(* CoDeSys 2.3.9.13 project: Stepper_03_Example02.pro *)
(* Libraries: D:\Daten\CodeSys_841\Projekte\Stepper\MC3\Release0.9.2\Stepper_03.lib 9.7.09 14:06:03, Standard.lib 22.11.04 11:21:12 *)

(* PLC configuration (modules and I/O channels)
Module Fieldbus Assignment [WAGO_Module] node 0, in %IB0 out %QB0 {INTTypePAAssignment = PLC; INTTypeModule = plugged}
Module Fieldbus Assignment [WAGO_Module] node 1, in %IB1 out %QB1 {INTTypePAAssignment = PLC; INTTypeModule = plugged}
Fieldbus variables [FB_VARS] node 1, in %IB0 out %QB0
*)

(* POU PLC_PRG, FBD *)
PROGRAM PLC_PRG
VAR

	myconfigtest673				:MC3_typConfiguration_673;

	Stepper1In AT%IB0			: ARRAY[0..11] OF BYTE;		(* input address stepper modul 750-673 *)
	Stepper1Out  AT%QB0 		: ARRAY[0..11] OF BYTE;		(* output address stepper modul 750-673 *)

	data1							: MC3_typData;
	MyCT							: MC3_ConfigurationTable;
	executeCT						: BOOL;
	readCT						: BOOL;
	writeCT						: BOOL;
	doneCT						: BOOL;
	busyCT						: BOOL;
	errorCT						: BOOL;
	statusCT						: WORD;

	MyDPT							: MC3_DriveProgramTable;
	executeDPT					: BOOL;
	readDPT						: BOOL;
	writeDPT						: BOOL;
	flashprogramDPT				: BOOL;
	dataCountDPT				: WORD:=14;
	doneDPT						: BOOL;
	busyDPT						: BOOL;
	errorDPT						: BOOL;
	statusDPT						: WORD;
	DataDPT		: ARRAY [0..MC3_gc_DriveProgramTableSize] OF BYTE:=
	(* opcode,  data_LSB, data, data_MSB  *)
		16#25, 16#20, 16#4E, 16#00,			(* set velocity  to 20.000 *)
		16#22, 16#B8, 16#0B, 16#00,			(* set acceleration to 3.000 *)
		16#04, 16#02, 16#00, 16#00,			(* Move_L to position 2 from position table*)
		16#70, 16#D0, 16#07, 16#00,			(* wait 2000 ms *)
		16#06, 16#88, 16#C3, 16#00,			(* Move relative 5.000 *)
		16#70, 16#D0, 16#07, 16#00,			(* wait 2000 ms *)
		16#06, 16#88, 16#C3, 16#00,			(* Move relative 5.000 *)
		16#70, 16#D0, 16#07, 16#00,			(* wait 2000 ms *)
		16#06, 16#88, 16#C3, 16#00,			(* Move relative 5.000 *)
		16#70, 16#D0, 16#07, 16#00,			(* wait 2000 ms *)
		16#25, 16#10, 16#27, 16#00,			(* set velocity to 10.000 *)
		16#02, 16#00, 16#00, 16#00,			(* move to position 0 *)
		16#02, 16#00, 16#00, 16#00,			(* move to position 0 *)
		16#F1, 16#00, 16#00, 16#00;			(* end, wenn das Fahrprogramm hiermit abgeschlossen wird, gibt es keinen Fehler am Ende *)

	PositionTable					: ARRAY [0..MC3_gc_PositionTableSize] OF BYTE:=
	(*  data_LSB, data, data_MSB  *)
		16#00, 16#10, 16#00, 16#00,			(* Position 0->8192 *)
		16#00, 16#20, 16#00, 16#00,			(* Position 1->16384 *)
		16#A0, 16#86, 16#01, 16#00,			(* Position 2->100.000*)
		16#C0, 16#D4, 16#01, 16#00;			(* Position 3->120.000*)
	executePT					: BOOL;
	readPT						: BOOL;
	writePT						: BOOL;
	dataCountPT				: BYTE:=4;


	donePT						: BOOL;
	busyPT						: BOOL;
	errorPT						: BOOL;
	statusPT						: WORD;

	MyJog672						: MC3_Jog_672;
	enableJOG					: BOOL;
	TimeoutJOG					: WORD;
	busyJOG						: BOOL;

	MyMoveRelative				: MC3_MoveRelative;
	executeMoveRelative			: BOOL;
	SpeedMoveRelative			: INT:=10000;
	AccelerationMoveRelative		: WORD:=32000;
	DecelerationMoveRelative	: WORD:=32000;
	PositionMoveRelative			: DINT:=100000;
	doneMoveRelative			: BOOL;
	busyMoveRelative				: BOOL;
	errorMoveRelative				: BOOL;


	MyMoveAbsolute				: MC3_MoveAbsolute;
	executeMoveAbsolute			: BOOL;
	SpeedMoveAbsolute			: INT:=10000;
	AccelerationMoveAbsolute	: WORD:=30000;
	PositionMoveAbsolute		: DINT:=20000;
	busyMoveAbsolute			: BOOL;
	doneMoveAbsolute			: BOOL;

	MyHoming						: MC3_Home;
	executeHoming				: BOOL;
	HomingPositive				: BOOL;
	HomingNegative				: BOOL;
	doneHoming					: BOOL;
	busyHoming					: BOOL;

	MyVelocity672					: MC3_MoveVelocity_672;
	executeMoveVelocity			: BOOL;
	SpeedMoveVelocity			: INT;
	AccelerationMoveVelocity		: WORD:=200;
	doneMoveVelocity				: BOOL;
	busyMoveVelocity				: BOOL;

	MyPower						: MC3_Power;
	enablePower					: BOOL;
	PowerEnabled				: BOOL;

	MyReadActualPosition		: MC3_ReadActualPosition;
	enableRead					: BOOL:=TRUE;
	PositionValid					: BOOL;
	ActualPosition					: DINT;
	ActualSpeed					: INT;
	ActualMode					: BYTE;
	MailboxActive					: BOOL;
	ModulReset					: BOOL;

	MyReset						: MC3_Reset;
	executeReset					: BOOL;
	doneReset					: BOOL;

	MyStop							: MC3_Stop;
	executeStop					: BOOL;
	doneStop						: BOOL;

	MyReadError					: MC3_ReadError;
	enableReadError				: BOOL;
	doneReadError				: BOOL;
	busyReadError				: BOOL;
	StepperError					: BOOL;
	status							: WORD;
	ErrorDescription				: MC3_error_codes;

	MySetPosition					: MC3_SetPosition;
	executeSet					: BOOL;
	positionSet					: DINT;
	doneSet						: BOOL;
	busySet						: BOOL;
	errorSet						: BOOL;

	MyDP							: MC3_DriveProgram;
	executeDP						: BOOL;
	startpositionDP				: WORD;
	doneDP						: BOOL;
	busyDP						: BOOL;
	actualpositionDP				: WORD;

	MyCV							: MC3_ConfigurationValue;
	executeCV						: BOOL;
	addressCV					: WORD;
	readwriteCV					: BYTE;
	valuesizeCV					: BYTE;
	valueCV						: DWORD;
	doneCV						: BOOL;
	busyCV						: BOOL;
	errorCV						: BOOL;
	statusCV						: WORD;



(*visualisation variables*)
	visu_enablePower:BOOL;
	visu_executeReset:BOOL;
	(*Basic_1: MC2_StepperControlBasic;
	BasicEnable: BOOL;
	BasicDone: BOOL;
	BasicJobType: MC2_Mode;
	BasicModule: WORD:=670;
	BasicPos: BOOL;
	BasicNeg: BOOL;
	BasicStop: BOOL;
	BasicSpeed: INT:=5000;
	BasicAcceleration: WORD:=10000;
	BasicDeceleration: WORD:=10000;
	BasicRefPosition: DINT:=100000;
	BasicStart: BOOL;
	BasicReset: BOOL;
	BasicBusy: BOOL;
	BasicActualPosition: DINT;
	BasicActualSpeed: INT;
	BasicMailboxActive: BOOL;
	BasicError: BOOL;
	BasicStatus: WORD;
	BasicErrorCodes: MC2_Error_Codes;*)
	startablauf: BOOL;
	ablaufstate: INT;

	count: INT;
	testcount: INT := 1;
	MyVelocity670: MC3_MoveVelocity_670;
	MyJog670: MC3_Jog_670;
	posJog: BOOL;
	negJog: BOOL;

	executeDefault: BOOL;
	doneDefault: BOOL;
	busyDefault: BOOL;
	errorDefault: BOOL;
	StatusDefault: WORD;
	Stepper_673: MC3_StepperCommunication;
	P3: MC3_Power;
	S3: MC3_Stop;
	R3: MC3_MoveRelative;
	M3: MC3_Home;
	Re3: MC3_Reset;
	Abs3: MC3_MoveAbsolute;
	MySetPosition3: MC3_SetPosition;
	MyReadActualPosition3: MC3_ReadActualPosition;
	MyReadError3: MC3_ReadError;
	MyCT3: MC3_ConfigurationTable;
	MyCV3: MC3_ConfigurationValue;
	MyVelocity672_3: MC3_MoveVelocity_672;
	MyJog670_3: MC3_Jog_672;
	jogTimeout: WORD;
	b1: MC3_StepperControlBasic;
	error: BOOL;
	TON1: TON;
	testwert1: DINT;
	Torque3: MC3_MoveTorque;
	doneTorque: BOOL;
	busyTorque: BOOL;
	executeTorque: BOOL;
	speedTorque: INT;
	currentTorque: WORD;
	Torque3_2: MC3_MoveTorque2;
	enableTorque: BOOL;
	doneTorque2: BOOL;
	busyTorque2: BOOL;
	MyDT: MC3_DriveProgramTable;
	MyPT: MC3_PositionTable;
	MyVelocity670_3: MC3_MoveVelocity_670;
	MyJog672_3: MC3_Jog_672;
END_VAR
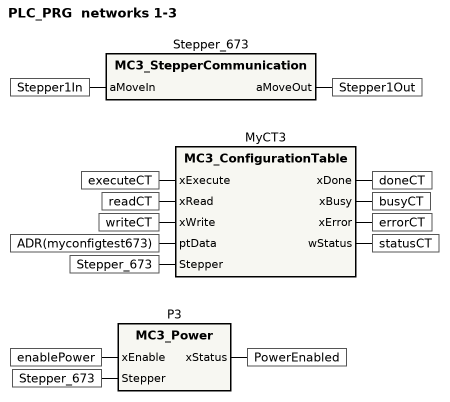
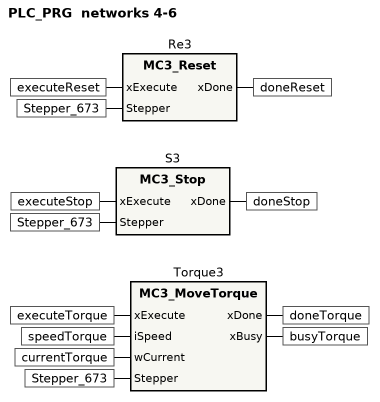
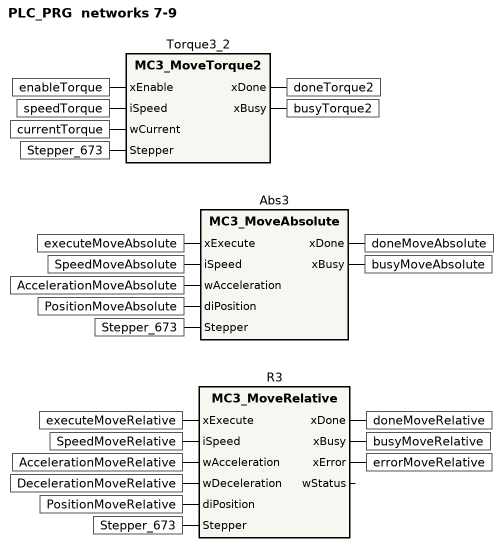
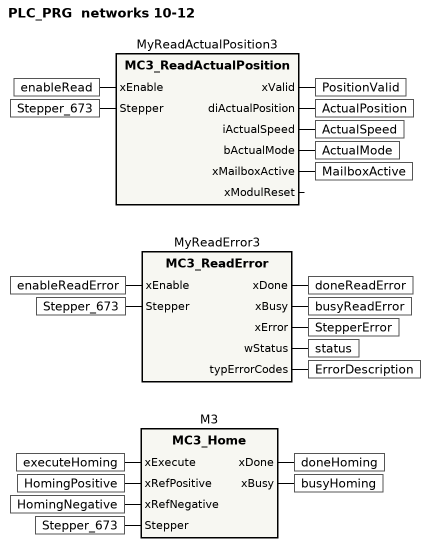
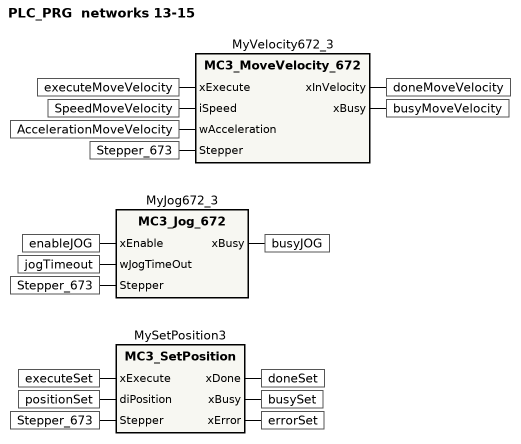
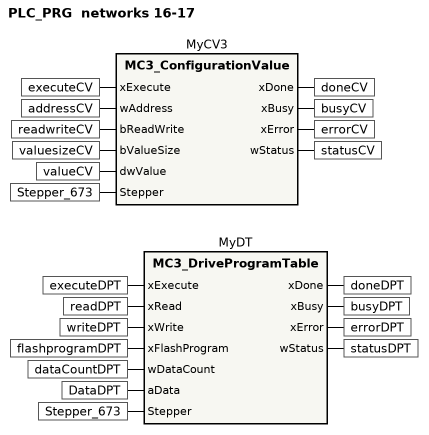
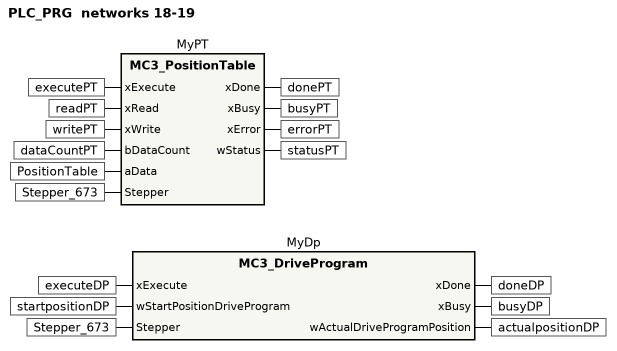
_FBD_ (* Function Block Diagram *)
NETWORK 1
	Stepper_673:MC3_StepperCommunication(aMoveIn: Stepper1In) => Stepper1Out
NETWORK 2
	MyCT3:MC3_ConfigurationTable(xExecute: executeCT, xRead: readCT, xWrite: writeCT, ptData: ADR(myconfigtest673), Stepper: Stepper_673, xBusy => busyCT, xError => errorCT, wStatus => statusCT) => doneCT
NETWORK 3
	P3:MC3_Power(xEnable: enablePower, Stepper: Stepper_673) => PowerEnabled
NETWORK 4
	Re3:MC3_Reset(xExecute: executeReset, Stepper: Stepper_673) => doneReset
NETWORK 5
	S3:MC3_Stop(xExecute: executeStop, Stepper: Stepper_673) => doneStop
NETWORK 6
	Torque3:MC3_MoveTorque(xExecute: executeTorque, iSpeed: speedTorque, wCurrent: currentTorque, Stepper: Stepper_673, xBusy => busyTorque) => doneTorque
NETWORK 7
	Torque3_2:MC3_MoveTorque2(xEnable: enableTorque, iSpeed: speedTorque, wCurrent: currentTorque, Stepper: Stepper_673, xBusy => busyTorque2) => doneTorque2
NETWORK 8
	Abs3:MC3_MoveAbsolute(xExecute: executeMoveAbsolute, iSpeed: SpeedMoveAbsolute, wAcceleration: AccelerationMoveAbsolute, diPosition: PositionMoveAbsolute, Stepper: Stepper_673, xBusy => busyMoveAbsolute) => doneMoveAbsolute
NETWORK 9
	R3:MC3_MoveRelative(xExecute: executeMoveRelative, iSpeed: SpeedMoveRelative, wAcceleration: AccelerationMoveRelative, wDeceleration: DecelerationMoveRelative, diPosition: PositionMoveRelative, Stepper: Stepper_673, xBusy => busyMoveRelative, xError => errorMoveRelative) => doneMoveRelative
NETWORK 10
	MyReadActualPosition3:MC3_ReadActualPosition(xEnable: enableRead, Stepper: Stepper_673, diActualPosition => ActualPosition, iActualSpeed => ActualSpeed, bActualMode => ActualMode, xMailboxActive => MailboxActive) => PositionValid
NETWORK 11
	MyReadError3:MC3_ReadError(xEnable: enableReadError, Stepper: Stepper_673, xBusy => busyReadError, xError => StepperError, wStatus => status, typErrorCodes => ErrorDescription) => doneReadError
NETWORK 12
	M3:MC3_Home(xExecute: executeHoming, xRefPositive: HomingPositive, xRefNegative: HomingNegative, Stepper: Stepper_673, xBusy => busyHoming) => doneHoming
NETWORK 13
	MyVelocity672_3:MC3_MoveVelocity_672(xExecute: executeMoveVelocity, iSpeed: SpeedMoveVelocity, wAcceleration: AccelerationMoveVelocity, Stepper: Stepper_673, xBusy => busyMoveVelocity) => doneMoveVelocity
NETWORK 14
	MyJog672_3:MC3_Jog_672(xEnable: enableJOG, wJogTimeOut: jogTimeout, Stepper: Stepper_673) => busyJOG
NETWORK 15
	MySetPosition3:MC3_SetPosition(xExecute: executeSet, diPosition: positionSet, Stepper: Stepper_673, xBusy => busySet, xError => errorSet) => doneSet
NETWORK 16
	MyCV3:MC3_ConfigurationValue(xExecute: executeCV, wAddress: addressCV, bReadWrite: readwriteCV, bValueSize: valuesizeCV, dwValue: valueCV, Stepper: Stepper_673, xBusy => busyCV, xError => errorCV, wStatus => statusCV) => doneCV
NETWORK 17
	MyDT:MC3_DriveProgramTable(xExecute: executeDPT, xRead: readDPT, xWrite: writeDPT, xFlashProgram: flashprogramDPT, wDataCount: dataCountDPT, aData: DataDPT, Stepper: Stepper_673, xBusy => busyDPT, xError => errorDPT, wStatus => statusDPT) => doneDPT
NETWORK 18
	MyPT:MC3_PositionTable(xExecute: executePT, xRead: readPT, xWrite: writePT, bDataCount: dataCountPT, aData: PositionTable, Stepper: Stepper_673, xBusy => busyPT, xError => errorPT, wStatus => statusPT) => donePT
NETWORK 19
	MyDp:MC3_DriveProgram(xExecute: executeDP, wStartPositionDriveProgram: startpositionDP, Stepper: Stepper_673, xBusy => busyDP, wActualDriveProgramPosition => actualpositionDP) => doneDP
_END_FBD_
(* the same logic as Structured Text *)
(* Network 1 *)
Stepper_673(aMoveIn := Stepper1In);
Stepper1Out := Stepper_673.aMoveOut;
(* Network 2 *)
MyCT3(xExecute := executeCT, xRead := readCT, xWrite := writeCT, ptData := ADR(myconfigtest673), Stepper := Stepper_673);
busyCT := MyCT3.xBusy;
errorCT := MyCT3.xError;
statusCT := MyCT3.wStatus;
doneCT := MyCT3.xDone;
(* Network 3 *)
P3(xEnable := enablePower, Stepper := Stepper_673);
PowerEnabled := P3.xStatus;
(* Network 4 *)
Re3(xExecute := executeReset, Stepper := Stepper_673);
doneReset := Re3.xDone;
(* Network 5 *)
S3(xExecute := executeStop, Stepper := Stepper_673);
doneStop := S3.xDone;
(* Network 6 *)
Torque3(xExecute := executeTorque, iSpeed := speedTorque, wCurrent := currentTorque, Stepper := Stepper_673);
busyTorque := Torque3.xBusy;
doneTorque := Torque3.xDone;
(* Network 7 *)
Torque3_2(xEnable := enableTorque, iSpeed := speedTorque, wCurrent := currentTorque, Stepper := Stepper_673);
busyTorque2 := Torque3_2.xBusy;
doneTorque2 := Torque3_2.xDone;
(* Network 8 *)
Abs3(xExecute := executeMoveAbsolute, iSpeed := SpeedMoveAbsolute, wAcceleration := AccelerationMoveAbsolute, diPosition := PositionMoveAbsolute, Stepper := Stepper_673);
busyMoveAbsolute := Abs3.xBusy;
doneMoveAbsolute := Abs3.xDone;
(* Network 9 *)
R3(xExecute := executeMoveRelative, iSpeed := SpeedMoveRelative, wAcceleration := AccelerationMoveRelative, wDeceleration := DecelerationMoveRelative, diPosition := PositionMoveRelative, Stepper := Stepper_673);
busyMoveRelative := R3.xBusy;
errorMoveRelative := R3.xError;
doneMoveRelative := R3.xDone;
(* Network 10 *)
MyReadActualPosition3(xEnable := enableRead, Stepper := Stepper_673);
ActualPosition := MyReadActualPosition3.diActualPosition;
ActualSpeed := MyReadActualPosition3.iActualSpeed;
ActualMode := MyReadActualPosition3.bActualMode;
MailboxActive := MyReadActualPosition3.xMailboxActive;
PositionValid := MyReadActualPosition3.xValid;
(* Network 11 *)
MyReadError3(xEnable := enableReadError, Stepper := Stepper_673);
busyReadError := MyReadError3.xBusy;
StepperError := MyReadError3.xError;
status := MyReadError3.wStatus;
ErrorDescription := MyReadError3.typErrorCodes;
doneReadError := MyReadError3.xDone;
(* Network 12 *)
M3(xExecute := executeHoming, xRefPositive := HomingPositive, xRefNegative := HomingNegative, Stepper := Stepper_673);
busyHoming := M3.xBusy;
doneHoming := M3.xDone;
(* Network 13 *)
MyVelocity672_3(xExecute := executeMoveVelocity, iSpeed := SpeedMoveVelocity, wAcceleration := AccelerationMoveVelocity, Stepper := Stepper_673);
busyMoveVelocity := MyVelocity672_3.xBusy;
doneMoveVelocity := MyVelocity672_3.xInVelocity;
(* Network 14 *)
MyJog672_3(xEnable := enableJOG, wJogTimeOut := jogTimeout, Stepper := Stepper_673);
busyJOG := MyJog672_3.xBusy;
(* Network 15 *)
MySetPosition3(xExecute := executeSet, diPosition := positionSet, Stepper := Stepper_673);
busySet := MySetPosition3.xBusy;
errorSet := MySetPosition3.xError;
doneSet := MySetPosition3.xDone;
(* Network 16 *)
MyCV3(xExecute := executeCV, wAddress := addressCV, bReadWrite := readwriteCV, bValueSize := valuesizeCV, dwValue := valueCV, Stepper := Stepper_673);
busyCV := MyCV3.xBusy;
errorCV := MyCV3.xError;
statusCV := MyCV3.wStatus;
doneCV := MyCV3.xDone;
(* Network 17 *)
MyDT(xExecute := executeDPT, xRead := readDPT, xWrite := writeDPT, xFlashProgram := flashprogramDPT, wDataCount := dataCountDPT, aData := DataDPT, Stepper := Stepper_673);
busyDPT := MyDT.xBusy;
errorDPT := MyDT.xError;
statusDPT := MyDT.wStatus;
doneDPT := MyDT.xDone;
(* Network 18 *)
MyPT(xExecute := executePT, xRead := readPT, xWrite := writePT, bDataCount := dataCountPT, aData := PositionTable, Stepper := Stepper_673);
busyPT := MyPT.xBusy;
errorPT := MyPT.xError;
statusPT := MyPT.wStatus;
donePT := MyPT.xDone;
(* Network 19 *)
MyDp(xExecute := executeDP, wStartPositionDriveProgram := startpositionDP, Stepper := Stepper_673);
busyDP := MyDp.xBusy;
actualpositionDP := MyDp.wActualDriveProgramPosition;
doneDP := MyDp.xDone;
END_PROGRAM
